PROGRAM Stn054_42_BufferRecircSpurMergePrestopGrn
VAR
	{attribute 'TcLinkToOSO' := '
			.iPuckPresent :=  <0,1,3>TIIB[N57S00 (AL1332)]^N57S03 (AL2341)^TxPDO^input byte 1;
			.iBufferFull  :=  <0,1,2>TIIB[N57S00 (AL1332)]^N57S03 (AL2341)^TxPDO^input byte 3;
			.oStopLower :=  <0,1,7>TIIB[N57S00 (AL1332)]^N57S02 (EX260)^RxPDO^output byte 1'}
	fbConvStop: FB_ConvStop;
END_VAR

//CleaningRecircMergeSpurPrestopGRN  (8B)
//GRN Buffer Recirc Merge Main Stop Puck Present
//GRN Buffer Recirc Merge Main DS Buffer
//GRN Buffer Recirc Merge Spur Puck Present

//
//  This code instantiates a component that is implimented as a common function block
//    Note that I/O is linked directly to I/O variables inside the named instance

gStn054_42_BufferRecircSpurMergePrestopGrn.ConvRunning  := gConsumed_SafetyInterfaceConv.MtrRunning.Enc058Mtr07 AND gConsumed_SafetyInterfaceConv.MtrRunning.Enc058Mtr06;

fbConvStop(
	pStn := ADR(gStn054),
	pCmp := ADR(gStn054_42_BufferRecircSpurMergePrestopGrn),
	pUpstreamStop := 0,
	pStateTraceBuffer := ADR(gStn054_StateTraceBuffer),
	pStateTraceFifo := ADR(gStn054_StateTraceFifo),
	pStats := ADR(gStn054_02_Stats));

END_PROGRAM

(* stored: Version 1.1.0.1, ProductVersion 3.1.4024.6
   POU Stn054_42_BufferRecircSpurMergePrestopGrn: Id {be925af1-ac0c-4ff8-9723-b1a48dd4ca89}, SpecialFunc None *)
